// TIA Portal project "FactoryIO_Template_S7-1200_V15_V15.1" (V15.1)
// Vorlageprojekt für das Buch mit Zielsystem S7-1200

(* hardware
DEVICE "S7-1200-Station_1"  S7-1200 Station
   slot 0: "Baugruppenträger_0"  Rack  V1.0
   slot 1: "PLC_1"  CPU 1211C DC/DC/DC  6ES7 211-1AE40-0XB0  V4.1
*)

// ===== PLC "PLC_1"  CPU 1211C DC/DC/DC =====

VAR_GLOBAL   // PLC tag table "Standard-Variablentabelle"
   "Entry_Conveyor" AT %A0.0 : Bool;
   "--" AT %E0.0 : Bool;
   "At_Load" AT %E0.1 : Bool;
   "Forks_Left" AT %Q0.2 : Bool;
   "At_Middle" AT %I0.3 : Bool;
   "Forks_Right" AT %Q0.3 : Bool;
   "Lift" AT %Q0.4 : Bool;
   "At_Right" AT %I0.4 : Bool;
   "Unload_Conveyor" AT %Q0.5 : Bool;
   "At_Unload" AT %I0.5 : Bool;
   "Exit_Conveyor" AT %Q0.6 : Bool;
   "Start_Light" AT %Q0.7 : Bool;
   "At_Exit" AT %I0.6 : Bool;
   "Reset_Light" AT %Q1.0 : Bool;
   "Moving_X" AT %I0.7 : Bool;
   "Stop_Light" AT %Q1.1 : Bool;
   "Moving_Z" AT %I1.0 : Bool;
   "Start" AT %I1.1 : Bool;
   "Reset" AT %I1.2 : Bool;
   "Stop" AT %I1.3 : Bool;
   "Emergency_stop" AT %I1.4 : Bool;
   "Auto" AT %I1.5 : Bool;
   "Running" AT %I1.6 : Bool;
   "is_on" AT %Q1.2 : Bool;
   "System_Byte" AT %MB1 : Byte;
   "FirstScan" AT %M1.0 : Bool;
   "DiagStatusUpdate" AT %M1.1 : Bool;
   "AlwaysTRUE" AT %M1.2 : Bool;
   "AlwaysFALSE" AT %M1.3 : Bool;
   "Clock_Byte" AT %MB0 : Byte;
   "Clock_10Hz" AT %M0.0 : Bool;
   "Clock_5Hz" AT %M0.1 : Bool;
   "Clock_2.5Hz" AT %M0.2 : Bool;
   "Clock_2Hz" AT %M0.3 : Bool;
   "Clock_1.25Hz" AT %M0.4 : Bool;
   "Clock_1Hz" AT %M0.5 : Bool;
   "Clock_0.625Hz" AT %M0.6 : Bool;
   "Clock_0.5Hz" AT %M0.7 : Bool;
   "M0_MoveToLift" AT %M100.0 : Bool;
   "M1_isAtLeft" AT %M100.1 : Bool;
   "M2_ReadyToLoad" AT %M100.2 : Bool;
   "M3_isLifted" AT %M100.3 : Bool;
   "M4_isLoaded" AT %M100.4 : Bool;
   "target_position" AT %QD30 : DWord;
   "M5_Positioned" AT %M100.5 : Bool;
   "M6_LiftedToUnload" AT %M100.6 : Bool;
   "M7_ReadyToUnload" AT %M100.7 : Bool;
   "M8_isUnloaded" AT %M200.0 : Bool;
   "number_filled" AT %QD31 : DWord;
   "Reset_position" AT %M200.1 : Bool;
   "Emergeny_is_pushed" AT %M200.2 : Bool;
END_VAR

VAR_GLOBAL   // PLC tag table "Tag table_1"
   "At_Left" AT %I0.2 : Bool;
   "Load_Conveyor" AT %Q0.1 : Bool;
END_VAR

// folder: System blocks/Program resources

DATA_BLOCK "IEC_Counter_0_DB"   // DB1
{ S7_Optimized_Access := 'TRUE' }
AUTHOR : Simatic
FAMILY : IEC
NAME : CNTR
VERSION : 1.0
// stored: InstanceOfName IEC_COUNTER
"IEC_COUNTER"
BEGIN
END_DATA_BLOCK

DATA_BLOCK "IEC_Timer_1_DB"   // DB3
{ S7_Optimized_Access := 'TRUE' }
AUTHOR : Simatic
FAMILY : IEC
NAME : IEC_TMR
VERSION : 1.0
// stored: InstanceOfName IEC_TIMER
"IEC_TIMER"
BEGIN
END_DATA_BLOCK

DATA_BLOCK "IEC_Timer_2_DB"   // DB4
{ S7_Optimized_Access := 'TRUE' }
AUTHOR : Simatic
FAMILY : IEC
NAME : IEC_TMR
VERSION : 1.0
// stored: InstanceOfName IEC_TIMER
"IEC_TIMER"
BEGIN
END_DATA_BLOCK

DATA_BLOCK "IEC_Timer_0_DB"   // DB5
{ S7_Optimized_Access := 'TRUE' }
AUTHOR : Simatic
FAMILY : IEC
NAME : IEC_TMR
VERSION : 1.0
// stored: InstanceOfName IEC_TIMER
"IEC_TIMER"
BEGIN
END_DATA_BLOCK

// folder: (top level)

FUNCTION "MHJ-PLC-Lab-Function-S71200" : Void   // FC9000, SCL
{ S7_Optimized_Access := 'TRUE' }
VERSION : 0.1
   VAR_TEMP
      rdTimeReturn : Int;
      outputTime : DTL;
      SyncVal : Byte;
      forVal : Int;
      forVal_2 : Int;
      Value : Byte;
   END_VAR
   VAR CONSTANT
      CompVal : Byte := 16#34;
      Value_01 : Byte := 16#11;
      Value_01_DW : DWord := 16#A165_D992;
      Value_02_DW : DWord := 16#58BE_4401;
   END_VAR
BEGIN

   #Value:=PEEK(area := 16#82,
        dbNumber := 0,
        byteOffset := 511);
   #Value := #Value + 1;

   POKE(area := 16#82,
        dbNumber := 0,
        byteOffset := 511,
        value := #Value);

   POKE(area:=16#81,
        dbNumber:=0,
        byteOffset:=1016,
        value:=#Value_01_DW);
   POKE(area := 16#81,
        dbNumber := 0,
        byteOffset := 1020,
        value := #Value_02_DW);

   POKE(area := 16#81,
        dbNumber := 0,
        byteOffset := 511,
        value := B#16#00);

   FOR #forVal := 0 TO 120 DO
       FOR #forVal_2:=0 TO 10 DO
           #rdTimeReturn:=RD_SYS_T(#outputTime);
           #rdTimeReturn := WR_SYS_T(#outputTime);
           #rdTimeReturn := RD_SYS_T(#outputTime);
           #rdTimeReturn := WR_SYS_T(#outputTime);
       END_FOR;
       #SyncVal:= PEEK(area := 16#81,
                      dbNumber := 0,
                      byteOffset := 511);
       IF #SyncVal = #CompVal THEN
          GOTO M_1;
       END_IF;
   END_FOR;
   RETURN;

   M_1:
   POKE(area := 16#81,
        dbNumber := 0,
        byteOffset := 511,
        value := B#16#0);
END_FUNCTION

ORGANIZATION_BLOCK "Main"   // OB1, FBD, ProgramCycle
TITLE = "Main Program Sweep (Cycle)"
{ S7_Optimized_Access := 'TRUE' }
VERSION : 0.1
   VAR_INPUT
      Initial_Call : Bool;   // Initial call of this OB
      Remanence : Bool;   // =True, if remanent data are available
   END_VAR
BEGIN

REGION Network 1: Konnektierungsbaustein für PLC-Lab
   // Im Netzwerk 1 wird der Konnektierungsbaustein für PLC-Lab aufgerufen.
   // Dieser Aufruf darf nicht entfernt werden!
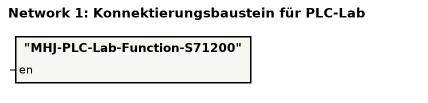
   "MHJ-PLC-Lab-Function-S71200"();
END_REGION

REGION Network 2: Ihr Programm
   // Schreiben Sie ab Netzwerk 2 Ihr Programm
END_REGION
END_ORGANIZATION_BLOCK

ORGANIZATION_BLOCK "Main_1"   // OB123, LAD, ProgramCycle
TITLE = "Main Program Sweep (Cycle)"
{ S7_Optimized_Access := 'TRUE' }
VERSION : 0.1
   VAR_INPUT
      Initial_Call : Bool;   // Initial call of this OB
      Remanence : Bool;   // =True, if remanent data are available
   END_VAR
   VAR_TEMP   // added for the SCL form of the ladder/FBD networks
      _w1 : Bool;
   END_VAR
BEGIN

REGION Network 1
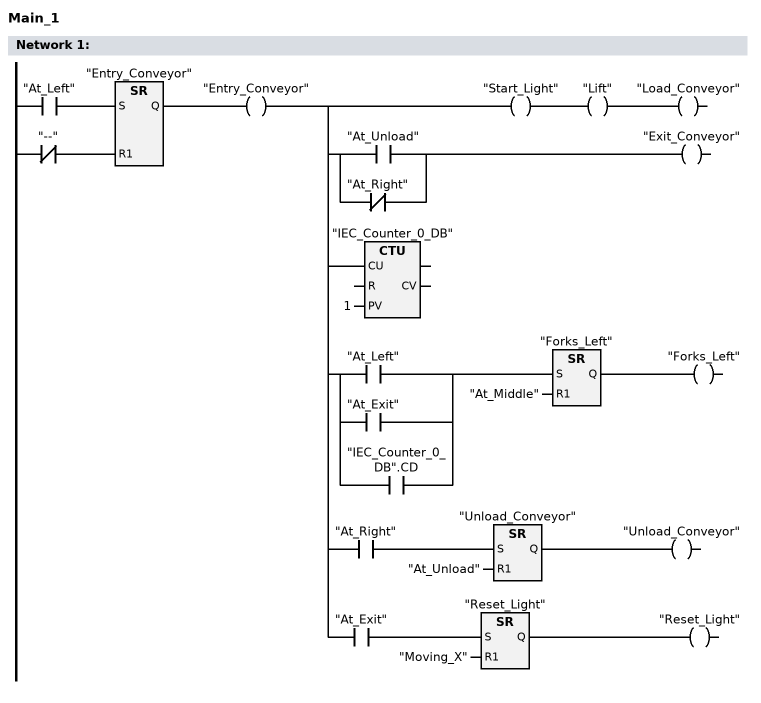
   IF "At_Left" THEN
       "Entry_Conveyor" := TRUE;   // SR flip-flop
   END_IF;
   IF NOT "--" THEN "Entry_Conveyor" := FALSE; END_IF;
   #_w1 := "Entry_Conveyor";
   "Entry_Conveyor" := #_w1;
   "Start_Light" := #_w1;
   "Lift" := #_w1;
   "Load_Conveyor" := #_w1;
   "Exit_Conveyor" := #_w1 AND ("At_Unload" OR NOT "At_Right");
   "IEC_Counter_0_DB".CTU(CU := #_w1, PV := 1);
   IF #_w1 AND ("At_Left" OR "At_Exit" OR "IEC_Counter_0_DB".CD) THEN
       "Forks_Left" := TRUE;   // SR flip-flop
   END_IF;
   IF "At_Middle" THEN "Forks_Left" := FALSE; END_IF;
   "Forks_Left" := "Forks_Left";
   IF #_w1 AND "At_Right" THEN
       "Unload_Conveyor" := TRUE;   // SR flip-flop
   END_IF;
   IF "At_Unload" THEN "Unload_Conveyor" := FALSE; END_IF;
   "Unload_Conveyor" := "Unload_Conveyor";
   IF #_w1 AND "At_Exit" THEN
       "Reset_Light" := TRUE;   // SR flip-flop
   END_IF;
   IF "Moving_X" THEN "Reset_Light" := FALSE; END_IF;
   "Reset_Light" := "Reset_Light";
END_REGION
END_ORGANIZATION_BLOCK

ORGANIZATION_BLOCK "Main_2"   // OB124, LAD, ProgramCycle
TITLE = "Main Program Sweep (Cycle)"
{ S7_Optimized_Access := 'TRUE' }
VERSION : 0.1
   VAR_INPUT
      Initial_Call : Bool;   // Initial call of this OB
      Remanence : Bool;   // =True, if remanent data are available
   END_VAR
   VAR_TEMP   // added for the SCL form of the ladder/FBD networks
      _w1 : Bool;
      _w2 : Bool;
      _w3 : Bool;
      _w4 : Bool;
      _w5 : Bool;
   END_VAR
BEGIN

REGION Network 1
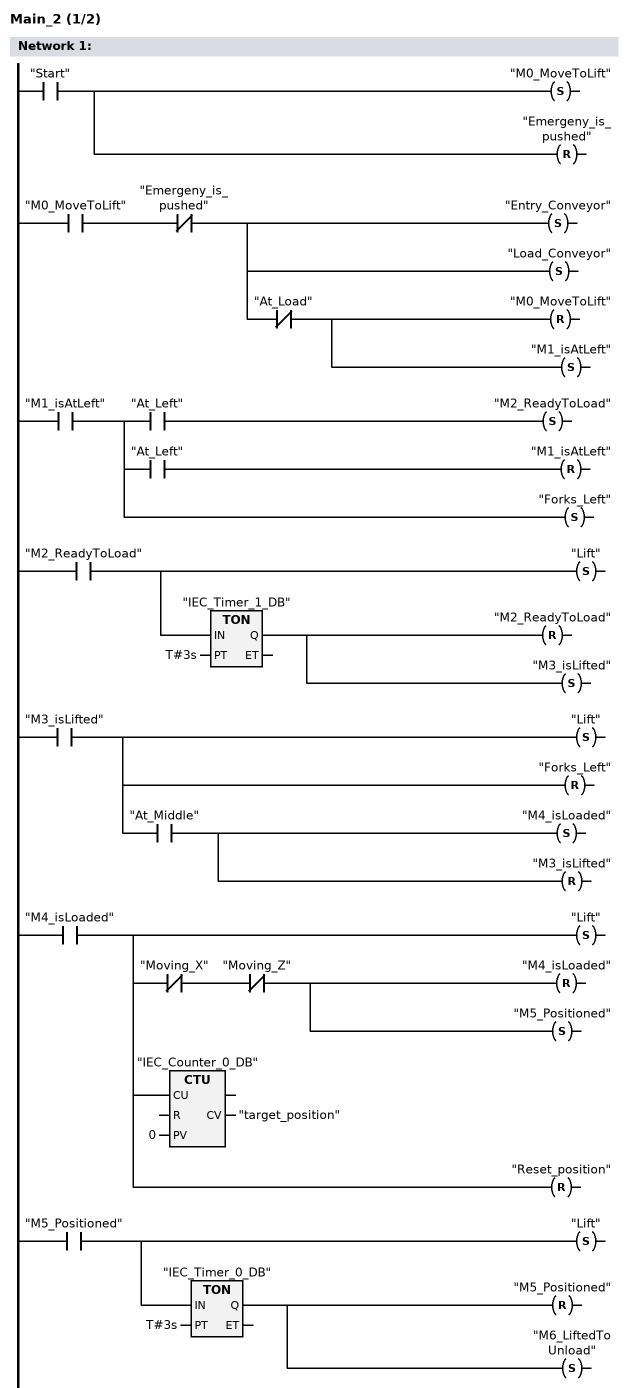
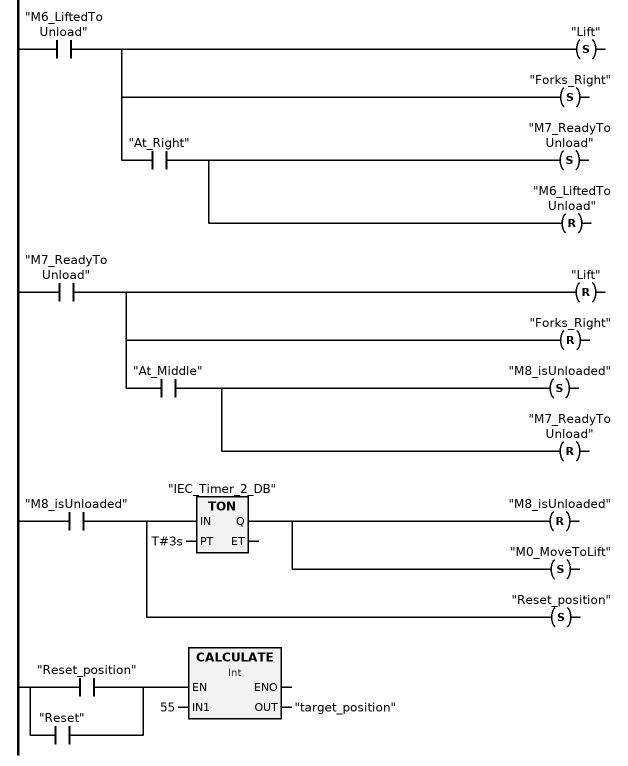
   IF "Start" THEN
       "M0_MoveToLift" := TRUE;
       "Emergeny_is_pushed" := FALSE;
   END_IF;
   #_w1 := "M0_MoveToLift" AND NOT "Emergeny_is_pushed";
   IF #_w1 THEN
       "Entry_Conveyor" := TRUE;
       "Load_Conveyor" := TRUE;
   END_IF;
   IF #_w1 AND NOT "At_Load" THEN
       "M0_MoveToLift" := FALSE;
       "M1_isAtLeft" := TRUE;
   END_IF;
   IF "M1_isAtLeft" AND "At_Left" THEN "M2_ReadyToLoad" := TRUE; END_IF;
   #_w2 := "M1_isAtLeft";
   IF "M1_isAtLeft" AND "At_Left" THEN "M1_isAtLeft" := FALSE; END_IF;
   IF #_w2 THEN "Forks_Left" := TRUE; END_IF;
   IF "M2_ReadyToLoad" THEN "Lift" := TRUE; END_IF;
   "IEC_Timer_1_DB".TON(IN := "M2_ReadyToLoad", PT := T#3s);
   IF "IEC_Timer_1_DB".Q THEN
       "M2_ReadyToLoad" := FALSE;
       "M3_isLifted" := TRUE;
   END_IF;
   IF "M3_isLifted" THEN
       "Lift" := TRUE;
       "Forks_Left" := FALSE;
   END_IF;
   IF "M3_isLifted" AND "At_Middle" THEN
       "M4_isLoaded" := TRUE;
       "M3_isLifted" := FALSE;
   END_IF;
   IF "M4_isLoaded" THEN "Lift" := TRUE; END_IF;
   #_w3 := "M4_isLoaded";
   #_w4 := "M4_isLoaded" AND NOT "Moving_X" AND NOT "Moving_Z";
   IF #_w4 THEN
       "M4_isLoaded" := FALSE;
       "M5_Positioned" := TRUE;
   END_IF;
   "IEC_Counter_0_DB".CTU(CU := #_w3, PV := 0, CV => "target_position");
   IF #_w3 THEN "Reset_position" := FALSE; END_IF;
   IF "M5_Positioned" THEN "Lift" := TRUE; END_IF;
   "IEC_Timer_0_DB".TON(IN := "M5_Positioned", PT := T#3s);
   IF "IEC_Timer_0_DB".Q THEN
       "M5_Positioned" := FALSE;
       "M6_LiftedToUnload" := TRUE;
   END_IF;
   IF "M6_LiftedToUnload" THEN
       "Lift" := TRUE;
       "Forks_Right" := TRUE;
   END_IF;
   IF "M6_LiftedToUnload" AND "At_Right" THEN
       "M7_ReadyToUnload" := TRUE;
       "M6_LiftedToUnload" := FALSE;
   END_IF;
   IF "M7_ReadyToUnload" THEN
       "Lift" := FALSE;
       "Forks_Right" := FALSE;
   END_IF;
   IF "M7_ReadyToUnload" AND "At_Middle" THEN
       "M8_isUnloaded" := TRUE;
       "M7_ReadyToUnload" := FALSE;
   END_IF;
   "IEC_Timer_2_DB".TON(IN := "M8_isUnloaded", PT := T#3s);
   #_w5 := "M8_isUnloaded";
   IF "IEC_Timer_2_DB".Q THEN
       "M8_isUnloaded" := FALSE;
       "M0_MoveToLift" := TRUE;
   END_IF;
   IF #_w5 THEN "Reset_position" := TRUE; END_IF;
   IF "Reset_position" OR "Reset" THEN "target_position" := 55; END_IF;
END_REGION

REGION Network 2
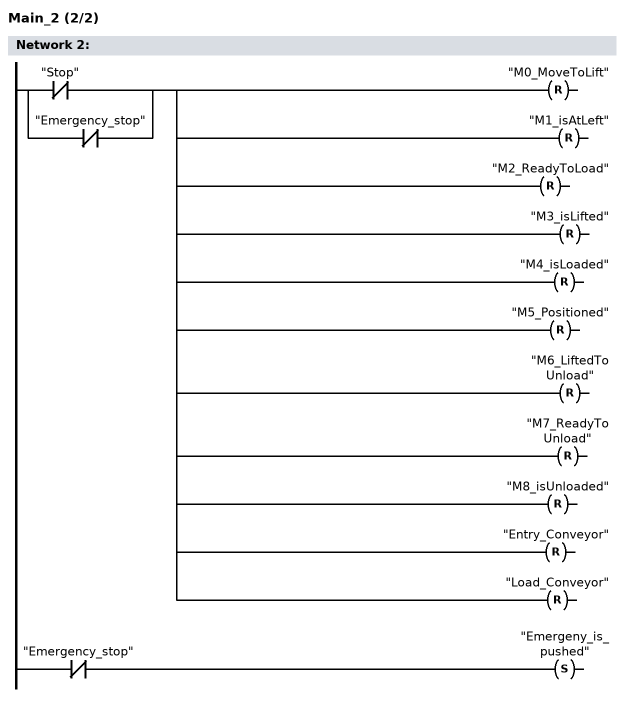
   RUNG wire#powerrail
      I_Contact( "Stop" )
      wire#w1
      R_Coil( "M0_MoveToLift" )
   END_RUNG
   RUNG wire#powerrail
      I_Contact( "Emergency_stop" )
   END_RUNG wire#w1
   RUNG wire#w1
      R_Coil( "M1_isAtLeft" )
   END_RUNG
   RUNG wire#w1
      R_Coil( "M2_ReadyToLoad" )
   END_RUNG
   RUNG wire#w1
      R_Coil( "M3_isLifted" )
   END_RUNG
   RUNG wire#w1
      R_Coil( "M4_isLoaded" )
   END_RUNG
   RUNG wire#w1
      R_Coil( "M5_Positioned" )
   END_RUNG
   RUNG wire#w1
      R_Coil( "M6_LiftedToUnload" )
   END_RUNG
   RUNG wire#w1
      R_Coil( "M7_ReadyToUnload" )
   END_RUNG
   RUNG wire#w1
      R_Coil( "M8_isUnloaded" )
   END_RUNG
   RUNG wire#w1
      R_Coil( "Entry_Conveyor" )
   END_RUNG
   RUNG wire#w1
      R_Coil( "Load_Conveyor" )
   END_RUNG
   RUNG wire#powerrail
      I_Contact( "Emergency_stop" )
      S_Coil( "Emergeny_is_pushed" )
   END_RUNG
   // the same network as SCL:
   IF NOT "Stop" OR NOT "Emergency_stop" THEN
       "M0_MoveToLift" := FALSE;
       "M1_isAtLeft" := FALSE;
       "M2_ReadyToLoad" := FALSE;
       "M3_isLifted" := FALSE;
       "M4_isLoaded" := FALSE;
       "M5_Positioned" := FALSE;
       "M6_LiftedToUnload" := FALSE;
       "M7_ReadyToUnload" := FALSE;
       "M8_isUnloaded" := FALSE;
       "Entry_Conveyor" := FALSE;
       "Load_Conveyor" := FALSE;
   END_IF;
   IF NOT "Emergency_stop" THEN "Emergeny_is_pushed" := TRUE; END_IF;
END_REGION
END_ORGANIZATION_BLOCK